# EPICS autosave request: iocBoot/ioc13cygwin/auto_positions.req
file "CARS_motor_positions.req",         P=13Cygwin:, M=m1
file "CARS_motor_positions.req",         P=13Cygwin:, M=m2
file "CARS_motor_positions.req",         P=13Cygwin:, M=m3
~
